{attribute addProperty BoxType "EL9576-0000-0016"}
{attribute addProperty Id "BCT_InputsAT %I*BCT_Inputs_BC823498120150WcStateAT %I*WcState_98A4DF7520.250InfoDataAT %I*InfoData_BC63D37F80100"}
{attribute addProperty CRC "3087002632"}
{attribute addProperty SizeInBites "202"}
{attribute addProperty SizeInBytes "25.25"}
TYPE EL9576_06679F76 :
STRUCT
	{attribute addProperty Name "BCT_Inputs"}
	BCT_Inputs : BCT_Inputs_BC823498;
	{attribute addProperty Name "WcState"}
	WcState : WcState_98A4DF75;
	{attribute addProperty Name "InfoData"}
	InfoData : InfoData_BC63D37F;
END_STRUCT
END_TYPE

(* stored: Version 1.2.0.0, ProductVersion 3.1.4024.9
   DUT EL9576_06679F76: Id {2a92fa53-f62d-42d7-a00e-5cb53dd22a6b} *)
